(* CODESYS project Mbc_Tc3_Pcs_v1.1.0.0.library
   Author: mbc engineering GmbH
   Placeholder: MBC TC3 PCS Library
   Title: MBC TC3 PCS Library
   Version: 1.1.0.0
   DocFormat: reStructuredText
   DefaultNamespace: Mbc_Tc3_Pcs
   Company: mbc engineering GmbH

Project tree, tasks and I/O mapping:
  Command/
    function block CommandBase [ST]: Abort, CalculateProgress, Call, Done, Init, Progress, SubTask, Task
    data type E_CommandResultCode
    interface ICommand: Call
    data type ST_CommandBaseHandshake
  docs/
    res/
      AddLibrary.JPG
    Changelog.md
    CommandBase.md
    Readme.md
  Version/
    global variables Global_Version
  Mbc_Tc3_Pcs.tmc
*)

// Command/E_CommandResultCode
// Default Result Code of the Command
{attribute 'qualified_only'}
{attribute 'strict'}
TYPE E_CommandResultCode :
(
	Init 			:= 0,
	Running 		:= 1,
	Done 			:= 2,
	Cancelled 		:= 3,
	StartCustom 	:= 100
) UINT;
END_TYPE

// Command/ST_CommandBaseHandshake
// Strukture for communication with PCS in the ``CommandBase`` class
TYPE ST_CommandBaseHandshake :
STRUCT
	bExecute		: BOOL;		// Will be set to true from the PCS to start the command. When the operation is finished, the PLC will it set to false. On a long running Task, the PCS can reset to false for Abort the operation. 
	bBusy			: BOOL;		// Is True when the command is executing.
	nResultCode		: UINT;		// Shows the operation result code of the commando state. Default Values see 'CommandResultCode' Enum Type. It is possible to set other codes!
	nProgress		: BYTE;		// Shows the optional calculated progress. The value is depend on the command implementation. (default can be 0..100%). Only necessary on long running operations.
	nSubTask		: UINT;		// Shows the optional state of long running Command Execution. It is possible to set it on own need.
END_STRUCT
END_TYPE

// Version/Global_Version
{attribute 'TcGenerated'}
// This function has been automatically generated from the project information.
VAR_GLOBAL CONSTANT
	{attribute 'const_non_replaced'}
	{attribute 'linkalways'}
	stLibVersion_MBC_TC3_PCS_Library : ST_LibVersion := (iMajor := 1, iMinor := 1, iBuild := 0, iRevision := 0, sVersion := '1.1.0.0');
END_VAR

// Command/CommandBase
// Basic implementation of a default command class for PCS interagtion with internal structure of ``ST_CommandBaseHandshake``.
// Aditional IN and OUT parameters should be declared in the derived implementation.
FUNCTION_BLOCK PUBLIC CommandBase IMPLEMENTS ICommand
VAR_IN_OUT
	(* Use Class Properties for IN_OUT Parameters!!! *)
END_VAR
VAR
	stHandshake		: ST_CommandBaseHandshake;		// Internal variable strukture for communication with PCS.
END_VAR

// OO-Class 
;

// Abort the ``Task`` Execution with the result code ``Cancelled``
METHOD PUBLIC Abort
Done(E_CommandResultCode.Cancelled);
END_METHOD

// Can be used to calculate the ``stHandshake.nProgress`` and ``stHandshake.nSubTask``
METHOD PROTECTED CalculateProgress
IF stHandshake.nResultCode = E_CommandResultCode.Done THEN
	stHandshake.nProgress := 100;
END_IF
END_METHOD

// The method is called in each cycle to execute the funktional part and the states of the command implementation.
METHOD PUBLIC Call
VAR
	bInit		: BOOL;
END_VAR
// Starting Case
stHandshake.bBusy S= bInit := (stHandshake.bExecute AND NOT stHandshake.bBusy);
IF bInit THEN
	stHandshake.nResultCode := E_CommandResultCode.Init;
	Init();
END_IF

// Cancel Case
IF NOT stHandshake.bExecute AND stHandshake.bBusy THEN
	Abort();
END_IF

// Running Case
IF stHandshake.bExecute AND stHandshake.bBusy THEN
	
	// Set Task init on First Call
	IF Task() THEN
		Done(E_CommandResultCode.Done);
	END_IF
		
	CalculateProgress();	
END_IF
END_METHOD

// Can be use to finish the ``Task`` Execution with a ``nResultCode``. 
METHOD PROTECTED Done
VAR_INPUT
	nResultCode		: UINT;
END_VAR
stHandshake.bBusy := stHandshake.bExecute := FALSE;
stHandshake.nResultCode := nResultCode;
END_METHOD

// Will be executed in the same cycle ``stHandshake.bExecute`` changes to ``true``
METHOD PROTECTED Init
VAR_INPUT
END_VAR
stHandshake.nResultCode := E_CommandResultCode.Running;
stHandshake.nProgress := 0;
stHandshake.nSubTask := 0;
END_METHOD

PROPERTY PROTECTED Progress : BYTE
GET
Progress := stHandshake.nProgress;
END_GET
SET
stHandshake.nProgress := Progress;
END_SET
END_PROPERTY

PROPERTY PROTECTED SubTask : UINT
GET
SubTask := stHandshake.nSubTask;
END_GET
SET
stHandshake.nSubTask := SubTask;
END_SET
END_PROPERTY

// Execute the funktional part of the command implementation. Will be executed in the same cycle ``stHandshake.bExecute`` changes to ``true`` after the ``Init`` Method
METHOD PROTECTED Task : BOOL
// Task complete if return true
Task := TRUE;
END_METHOD

END_FUNCTION_BLOCK

// Command/ICommand
// Minimal Command interface
INTERFACE ICommand

// The method is called in each cycle to execute the funktional part and the states of the command implementation.
METHOD Call
END_METHOD

END_INTERFACE
